FUNCTION_BLOCK TagOwner IMPLEMENTS I_TagOwner;

PROPERTY Self : I_TagOwner
GET
Self := THIS^;
END_GET
END_PROPERTY

END_FUNCTION_BLOCK

(* stored: Version 1.1.0.1
   POU TagOwner: Id {9c425f65-2eaa-48f8-ae7a-4e0b35161a36}, SpecialFunc None
   Property Self: Id {e4e76ef9-3c31-481e-89f1-7110d535e1cb}
   Get Get: Id {9359da33-4dcd-43b7-bcc6-ebeebb11763b} *)
